Omron Sysmac Studio project RingBufferOpcUaExtensionLib (Sysmac Studio 1.63.0.7, LibraryProject)
(* Develop extension library for operating RingBuffer via OPC UA. *)

# Controller LIB: NX102-9000 version 1.64
Task Services (priority 18, period or condition 4000): ModelTest
Library RingBufferLib 0.0.2 (contents left out)

PROGRAM README
RETURN;
(*

# About this project
This project is for the development of `RingBufferOpcUaExtensionLib`.
`RingBufferOpcUaExtensionLib` exposes a **RingBuffer** using the FB instance publication of the OPC UA server.
The exposed **RingBuffer** can be used like an RPC with an appropriate OPC UA client and proper operating procedures.

## About programs

* POU/Program/ModelTest
  This is a test program for clients that use the exposed **RingBuffer**.


# このプロジェクトについて
このプロジェクトは、`RingBufferOpcUaExtensionLib`の開発用プロジェクトです。
`RingBufferOpcUaExtensionLib`は、OPC UAサーバのFBインスタンス公開を使用して`RingBuffer`を公開します。
公開した`RingBuffer`は、適切なOPC UAクライアントと操作手順によりRPCのように使用できるようになります。

## プログラムについて

* POU/プログラム/ModelTest
  公開した`RingBuffer`を使用するクライアント用のテストプログラムです。


For the parts to which I have rights, I follow POU/Program/LICENSE.
You are free to use and modify it, but we are not responsible for any damage or loss related to it.

(c) 2025 KITA Munemitsu

*)
END_PROGRAM

PROGRAM ModelTest
VAR
    ModelTestOpcUaRingBuffer : ModelTest_OpcUaRingBuffer;
END_VAR
IF P_First_Run THEN
	ModelTestOpcUaRingBuffer.Enable := TRUE;
END_IF;

ModelTestOpcUaRingBuffer();
END_PROGRAM

PROGRAM LICENSE
RETURN;
(*
The MIT License (MIT)

Copyright(c) 2025 KITA Munemitsu

Permission is hereby granted, free of charge, to any person obtaining a copy of this software and associated
documentation files (the “Software”), to deal in the Software without restriction, including without limitation
the rights to use, copy, modify, merge, publish, distribute, sublicense, and/or sell copies of the Software,
and to permit persons to whom the Software is furnished to do so, subject to the following conditions:

The above copyright notice and this permission notice shall be included in all copies or substantial portions of the Software.

THE SOFTWARE IS PROVIDED “AS IS”, WITHOUT WARRANTY OF ANY KIND, EXPRESS OR IMPLIED, INCLUDING BUT NOT
LIMITED TO THE WARRANTIES OF MERCHANTABILITY, FITNESS FOR A PARTICULAR PURPOSE AND NONINFRINGEMENT.
IN NO EVENT SHALL THE AUTHORS OR COPYRIGHT HOLDERS BE LIABLE FOR ANY CLAIM, DAMAGES OR OTHER LIABILITY,
WHETHER IN AN ACTION OF CONTRACT, TORT OR OTHERWISE, ARISING FROM, OUT OF OR IN CONNECTION WITH THE SOFTWARE
OR THE USE OR OTHER DEALINGS IN THE SOFTWARE.
*)
END_PROGRAM

FUNCTION_BLOCK stfreakjp\buf\extension\OpcUaRingBuffer
VAR
    Read : stfreakjp\buf\extension\OpcUaRingBuffer_read;
    ReadFully : stfreakjp\buf\extension\OpcUaRingBuffer_readFully;
    Peek : stfreakjp\buf\extension\OpcUaRingBuffer_peek;
    PeekFully : stfreakjp\buf\extension\OpcUaRingBuffer_peekFully;
    Write : stfreakjp\buf\extension\OpcUaRingBuffer_write;
    WriteFully : stfreakjp\buf\extension\OpcUaRingBuffer_writeFully;
    Consume : stfreakjp\buf\extension\OpcUaRingBuffer_consume;
    ClearBuffer : stfreakjp\buf\extension\OpcUaRingBuffer_clear;
    GetReadableSize : stfreakjp\buf\extension\OpcUaRingBuffer_getReadableSize;
    GetWritableSize : stfreakjp\buf\extension\OpcUaRingBuffer_getWritableSize;
    GetStat : stfreakjp\buf\extension\OpcUaRingBuffer_getStat;
    IsOverflow : stfreakjp\buf\extension\OpcUaRingBuffer_isOverflow;
    IsReadable : stfreakjp\buf\extension\OpcUaRingBuffer_isReadable;
    IsWritable : stfreakjp\buf\extension\OpcUaRingBuffer_isWritable;
    GetContext : stfreakjp\buf\extension\OpcUaRingBuffer_getContext;
    DiffWrite : stfreakjp\buf\extension\OpcUaRingBuffer_diffWrite;
    DiffRead : stfreakjp\buf\extension\OpcUaRingBuffer_diffRead;
    Diff : stfreakjp\buf\extension\OpcUaRingBuffer_diff;
    GetDiffStat : stfreakjp\buf\extension\OpcUaRingBuffer_getDiffStat;
END_VAR
VAR_INPUT
    Enable : BOOL;
END_VAR
VAR_IN_OUT
    BufferContext : stfreakjp\buf\RingBufferContext;
    Buffer : ARRAY[*] OF BYTE;
END_VAR
VAR_OUTPUT
    Busy : BOOL;
END_VAR
IF NOT (Enable OR Busy) THEN
	RETURN;
END_IF;

IF Enable <> Busy THEN
	Read.Execute := FALSE;
	ReadFully.Execute := FALSE;
	Peek.Execute := FALSE;
	PeekFully.Execute := FALSE;
	Write.Execute := FALSE;
	WriteFully.Execute := FALSE;
	Consume.Execute := FALSE;
	ClearBuffer.Execute := FALSE;
	GetReadableSize.Execute := FALSE;
	GetWritableSize.Execute := FALSE;
	GetStat.Execute := FALSE;
	IsOverflow.Execute := FALSE;
	IsReadable.Execute := FALSE;
	IsWritable.Execute := FALSE;
	
	GetContext.Execute := FALSE;
	DiffWrite.Execute := FALSE;
	DiffRead.Execute := FALSE;
	Diff.Execute := FALSE;
	GetDiffStat.Execute := FALSE;
END_IF;
Busy := Enable;

Read(BufferContext:=BufferContext, Buffer:=Buffer);
ReadFully(BufferContext:=BufferContext, Buffer:=Buffer);
Peek(BufferContext:=BufferContext, Buffer:=Buffer);
PeekFully(BufferContext:=BufferContext, Buffer:=Buffer);
Write(BufferContext:=BufferContext, Buffer:=Buffer);
WriteFully(BufferContext:=BufferContext, Buffer:=Buffer);
Consume(BufferContext:=BufferContext, Buffer:=Buffer);
ClearBuffer(BufferContext:=BufferContext, Buffer:=Buffer);
GetReadableSize(BufferContext:=BufferContext);
GetWritableSize(BufferContext:=BufferContext);
GetStat(BufferContext:=BufferContext);
IsOverflow(BufferContext:=BufferContext);
IsReadable(BufferContext:=BufferContext);
IsWritable(BufferContext:=BufferContext);
	
GetContext(BufferContext:=BufferContext);
DiffWrite(BufferContext:=BufferContext, Buffer:=Buffer);
DiffRead(BufferContext:=BufferContext, Buffer:=Buffer);
Diff(BufferContext:=BufferContext, Buffer:=Buffer);
GetDiffStat(BufferContext:=BufferContext);
END_FUNCTION_BLOCK

FUNCTION_BLOCK stfreakjp\buf\extension\OpcUaRingBuffer_read
VAR_INPUT
    Execute : BOOL := False;
END_VAR
VAR_IN_OUT
    BufferContext : stfreakjp\buf\RingBufferContext;
    Buffer : ARRAY[*] OF BYTE;
END_VAR
VAR_INPUT
    Size : UINT := 0;
END_VAR
VAR_OUTPUT
    Out : ARRAY[0..8191] OF BYTE;
    ReadSize : UINT;
    Overflow : BOOL;
    Done : BOOL;
END_VAR
IF NOT Execute THEN
	IF Done THEN
		ReadSize := 0;
		Overflow := FALSE;
		Done := FALSE;
	END_IF;
	
	RETURN;
END_IF;

IF Execute AND NOT Done THEN
	\\stfreakjp\buf\RingBuffer_read(
						Context:=BufferContext,
						Buffer:=Buffer,
						Size:=Size,
						Out:=Out,
						Head:=0,
						ReadSize=>ReadSize,
						Overflow=>Overflow);
	Done := TRUE;
END_IF;
END_FUNCTION_BLOCK

FUNCTION_BLOCK stfreakjp\buf\extension\OpcUaRingBuffer_readFully
VAR_INPUT
    Execute : BOOL;
END_VAR
VAR_IN_OUT
    BufferContext : stfreakjp\buf\RingBufferContext;
    Buffer : ARRAY[*] OF BYTE;
END_VAR
VAR_OUTPUT
    Out : ARRAY[0..8191] OF BYTE;
    ReadSize : UINT;
    Overflow : BOOL;
    Done : BOOL;
END_VAR
IF NOT Execute THEN
	IF Done THEN
		ReadSize := 0;
		Overflow := FALSE;
		Done := FALSE;
	END_IF;
	
	RETURN;
END_IF;

IF Execute AND NOT Done THEN
	\\stfreakjp\buf\RingBuffer_readFully(
						Context:=BufferContext,
						Buffer:=Buffer,
						Out:=Out,
						Head:=0,
						ReadSize=>ReadSize,
						Overflow=>Overflow);
	Done := TRUE;
END_IF;
END_FUNCTION_BLOCK

FUNCTION_BLOCK stfreakjp\buf\extension\OpcUaRingBuffer_peek
VAR_INPUT
    Execute : BOOL := False;
END_VAR
VAR_IN_OUT
    BufferContext : stfreakjp\buf\RingBufferContext;
    Buffer : ARRAY[*] OF BYTE;
END_VAR
VAR_INPUT
    Size : UINT := 0;
END_VAR
VAR_OUTPUT
    Out : ARRAY[0..8191] OF BYTE;
    ReadSize : UINT;
    Overflow : BOOL;
    Done : BOOL;
END_VAR
IF NOT Execute THEN
	IF Done THEN
		ReadSize := 0;
		Overflow := FALSE;
		Done := FALSE;
	END_IF;
	
	RETURN;
END_IF;

IF Execute AND NOT Done THEN
	\\stfreakjp\buf\RingBuffer_peek(
						Context:=BufferContext,
						Buffer:=Buffer,
						Size:=Size,
						Out:=Out,
						Head:=0,
						ReadSize=>ReadSize,
						Overflow=>Overflow);
	Done := TRUE;
END_IF;
END_FUNCTION_BLOCK

FUNCTION_BLOCK stfreakjp\buf\extension\OpcUaRingBuffer_peekFully
VAR_INPUT
    Execute : BOOL := False;
END_VAR
VAR_IN_OUT
    BufferContext : stfreakjp\buf\RingBufferContext;
    Buffer : ARRAY[*] OF BYTE;
END_VAR
VAR_OUTPUT
    Out : ARRAY[0..8191] OF BYTE;
    ReadSize : UINT;
    Overflow : BOOL;
    Done : BOOL;
END_VAR
IF NOT Execute THEN
	IF Done THEN
		ReadSize := 0;
		Overflow := FALSE;
		Done := FALSE;
	END_IF;
	
	RETURN;
END_IF;

IF Execute AND NOT Done THEN
	\\stfreakjp\buf\RingBuffer_peekFully(
						Context:=BufferContext,
						Buffer:=Buffer,
						Out:=Out,
						Head:=0,
						ReadSize=>ReadSize,
						Overflow=>Overflow);
	Done := TRUE;
END_IF;
END_FUNCTION_BLOCK

FUNCTION_BLOCK stfreakjp\buf\extension\OpcUaRingBuffer_write
VAR
    iTmpIn : ARRAY[0..8191] OF BYTE;
END_VAR
VAR_INPUT
    Execute : BOOL := False;
END_VAR
VAR_IN_OUT
    BufferContext : stfreakjp\buf\RingBufferContext;
    Buffer : ARRAY[*] OF BYTE;
END_VAR
VAR_INPUT
    In : ARRAY[0..8191] OF BYTE;
    Size : UINT := 0;
    AllowOverwrite : BOOL;
END_VAR
VAR_OUTPUT
    Ok : BOOL;
    Done : BOOL;
END_VAR
IF NOT Execute THEN
	Done := FALSE;

	RETURN;
END_IF;

IF Execute AND NOT Done THEN
	MemCopy(In:=In[0], AryOut:=iTmpIn[0], Size:=Size);	
	Ok := \\stfreakjp\buf\RingBuffer_write(
							  Context:=BufferContext,
							  Buffer:=Buffer,
							  In:=iTmpIn,
							  Head:=0,
							  Size:=Size,
							  AllowOverwrite:=AllowOverwrite);
	Done := TRUE;
END_IF;
END_FUNCTION_BLOCK

FUNCTION_BLOCK stfreakjp\buf\extension\OpcUaRingBuffer_writeFully
VAR
    iTmpIn : ARRAY[0..8191] OF BYTE;
END_VAR
VAR_INPUT
    Execute : BOOL := False;
END_VAR
VAR_IN_OUT
    BufferContext : stfreakjp\buf\RingBufferContext;
    Buffer : ARRAY[*] OF BYTE;
END_VAR
VAR_INPUT
    In : ARRAY[0..8191] OF BYTE;
    Size : UINT := 0;
END_VAR
VAR_OUTPUT
    WriteSize : UINT;
    Done : BOOL;
END_VAR
IF NOT Execute THEN
	IF Done THEN
		WriteSize := 0;
		Done := FALSE;
	END_IF;

	RETURN;
END_IF;

IF Execute AND NOT Done THEN
	MemCopy(In:=In[0], AryOut:=iTmpIn[0], Size:=Size);	
	\\stfreakjp\buf\RingBuffer_writeFully(
						Context:=BufferContext,
						Buffer:=Buffer,
						In:=iTmpIn,
						Head:=0,
						Size:=Size,
						WriteSize=>WriteSize);
	Done := TRUE;
END_IF;
END_FUNCTION_BLOCK

FUNCTION_BLOCK stfreakjp\buf\extension\OpcUaRingBuffer_consume
VAR_INPUT
    Execute : BOOL := False;
END_VAR
VAR_IN_OUT
    BufferContext : stfreakjp\buf\RingBufferContext;
    Buffer : ARRAY[*] OF BYTE;
END_VAR
VAR_INPUT
    Size : UINT := 0;
END_VAR
VAR_OUTPUT
    Ok : BOOL;
    Done : BOOL;
END_VAR
IF NOT Execute THEN
	Done := FALSE;
	
	RETURN;
END_IF;

IF Execute AND NOT Done THEN
	Ok := \\stfreakjp\buf\RingBuffer_consume(
							  Context:=BufferContext,
							  Buffer:=Buffer,
							  Size:=Size);
	Done := TRUE;
END_IF;
END_FUNCTION_BLOCK

FUNCTION_BLOCK stfreakjp\buf\extension\OpcUaRingBuffer_clear
VAR_INPUT
    Execute : BOOL := False;
END_VAR
VAR_IN_OUT
    BufferContext : stfreakjp\buf\RingBufferContext;
    Buffer : ARRAY[*] OF BYTE;
END_VAR
VAR_OUTPUT
    Ok : BOOL;
    Done : BOOL;
END_VAR
IF NOT Execute THEN
	Done := FALSE;
	
	RETURN;
END_IF;

IF Execute AND NOT Done THEN
	Ok := \\stfreakjp\buf\RingBuffer_clear(
							  Context:=BufferContext,
							  Buffer:=Buffer);
	Done := TRUE;
END_IF;
END_FUNCTION_BLOCK

FUNCTION_BLOCK stfreakjp\buf\extension\OpcUaRingBuffer_getReadableSize
VAR_INPUT
    Execute : BOOL := False;
END_VAR
VAR_IN_OUT
    BufferContext : stfreakjp\buf\RingBufferContext;
END_VAR
VAR_OUTPUT
    Size : UINT;
    Done : BOOL;
END_VAR
IF NOT Execute THEN
	IF Done THEN
		Size := 0;
		Done := FALSE;
	END_IF;
	
	RETURN;
END_IF;

IF Execute AND NOT Done THEN
	\\stfreakjp\buf\RingBuffer_getReadableSize(
						Context:=BufferContext,
						Size=>Size);
	Done := TRUE;
END_IF;
END_FUNCTION_BLOCK

FUNCTION_BLOCK stfreakjp\buf\extension\OpcUaRingBuffer_getWritableSize
VAR_INPUT
    Execute : BOOL;
END_VAR
VAR_IN_OUT
    BufferContext : stfreakjp\buf\RingBufferContext;
END_VAR
VAR_OUTPUT
    Size : UINT;
    Done : BOOL;
END_VAR
IF NOT Execute THEN
	IF Done THEN
		Size := 0;
		Done := FALSE;
	END_IF;
	
	RETURN;
END_IF;

IF Execute AND NOT Done THEN
	\\stfreakjp\buf\RingBuffer_getWritableSize(
						Context:=BufferContext,
						Size=>Size);
	Done := TRUE;
END_IF;
END_FUNCTION_BLOCK

FUNCTION_BLOCK stfreakjp\buf\extension\OpcUaRingBuffer_getStat
VAR_INPUT
    Execute : BOOL;
END_VAR
VAR_IN_OUT
    BufferContext : stfreakjp\buf\RingBufferContext;
END_VAR
VAR_OUTPUT
    WritableSize : UINT;
    ReadableSize : UINT;
    Overflow : BOOL;
    Done : BOOL;
END_VAR
IF NOT Execute THEN
	IF Done THEN
		WritableSize := 0;
		ReadableSize := 0;
		Overflow := FALSE;
		Done := FALSE;
	END_IF;
	
	RETURN;
END_IF;

IF Execute AND NOT Done THEN
	\\stfreakjp\buf\RingBuffer_getStat(
						Context:=BufferContext,
						WritableSize=>WritableSize,
						ReadableSize=>ReadableSize,
						Overflow=>Overflow);
	Done := TRUE;
END_IF;
END_FUNCTION_BLOCK

FUNCTION_BLOCK stfreakjp\buf\extension\OpcUaRingBuffer_isOverflow
VAR_INPUT
    Execute : BOOL;
END_VAR
VAR_IN_OUT
    BufferContext : stfreakjp\buf\RingBufferContext;
END_VAR
VAR_OUTPUT
    Overflow : BOOL;
    Done : BOOL;
END_VAR
IF NOT Execute THEN
	Overflow := FALSE;
	Done := FALSE;
	
	RETURN;
END_IF;

IF Execute AND NOT Done THEN
	Overflow := \\stfreakjp\buf\RingBuffer_isOverflow(
									Context:=BufferContext);
	Done := TRUE;
END_IF;
END_FUNCTION_BLOCK

FUNCTION_BLOCK stfreakjp\buf\extension\OpcUaRingBuffer_isReadable
VAR_INPUT
    Execute : BOOL;
END_VAR
VAR_IN_OUT
    BufferContext : stfreakjp\buf\RingBufferContext;
END_VAR
VAR_OUTPUT
    Readable : BOOL;
    Done : BOOL;
END_VAR
IF NOT Execute THEN
	Readable := FALSE;
	Done := FALSE;
	
	RETURN;
END_IF;

IF Execute AND NOT Done THEN
	Readable := \\stfreakjp\buf\RingBuffer_isReadable(
									Context:=BufferContext);
	Done := TRUE;
END_IF;
END_FUNCTION_BLOCK

FUNCTION_BLOCK stfreakjp\buf\extension\OpcUaRingBuffer_isWritable
VAR_INPUT
    Execute : BOOL;
END_VAR
VAR_IN_OUT
    BufferContext : stfreakjp\buf\RingBufferContext;
END_VAR
VAR_OUTPUT
    Writable : BOOL;
    Done : BOOL;
END_VAR
IF NOT Execute THEN
	Writable := FALSE;
	Done := FALSE;
	
	RETURN;
END_IF;

IF Execute AND NOT Done THEN
	Writable := \\stfreakjp\buf\RingBuffer_isWritable(
									Context:=BufferContext);
	Done := TRUE;
END_IF;
END_FUNCTION_BLOCK

FUNCTION_BLOCK stfreakjp\buf\extension\OpcUaRingBuffer_getContext
VAR_INPUT
    Execute : BOOL;
END_VAR
VAR_IN_OUT
    BufferContext : stfreakjp\buf\RingBufferContext;
END_VAR
VAR_OUTPUT
    Context : stfreakjp\buf\RingBufferContext;
    Done : BOOL;
END_VAR
IF NOT Execute THEN
	IF Done THEN
		Clear(Context);
		Done := FALSE;
	END_IF;
	
	RETURN;
END_IF;

IF Execute AND NOT Done THEN
	Context := BufferContext;
	Done := TRUE;
END_IF;
END_FUNCTION_BLOCK

FUNCTION_BLOCK stfreakjp\buf\extension\OpcUaRingBuffer_diffWrite
VAR
    iRefContext : stfreakjp\buf\RingBufferContext;
END_VAR
VAR_INPUT
    Execute : BOOL;
END_VAR
VAR_IN_OUT
    BufferContext : stfreakjp\buf\RingBufferContext;
    Buffer : ARRAY[*] OF BYTE;
END_VAR
VAR_INPUT
    RefContext : stfreakjp\buf\RingBufferContext;
END_VAR
VAR_OUTPUT
    Out : ARRAY[0..8191] OF BYTE;
    Size : UINT;
    Missing : BOOL;
    ComparedContext : stfreakjp\buf\RingBufferContext;
    Done : BOOL;
END_VAR
IF NOT Execute THEN
	IF Done THEN
		Size := 0;
		Missing := FALSE;
		Clear(ComparedContext);
		Done := FALSE;
	END_IF;
	
	RETURN;
END_IF;

IF Execute AND NOT Done THEN
	iRefContext := RefContext;
	\\stfreakjp\buf\RingBuffer_diffWrite(
						Context:=BufferContext,
						Buffer:=Buffer,
						RefContext:=iRefContext,
						Diff:=Out,
						Head:=0,
						Size=>Size,
						Missing=>Missing,
						ComparedContext=>ComparedContext);
	Done := TRUE;
END_IF;
END_FUNCTION_BLOCK

FUNCTION_BLOCK stfreakjp\buf\extension\OpcUaRingBuffer_diffRead
VAR
    iRefContext : stfreakjp\buf\RingBufferContext;
END_VAR
VAR_INPUT
    Execute : BOOL;
END_VAR
VAR_IN_OUT
    BufferContext : stfreakjp\buf\RingBufferContext;
    Buffer : ARRAY[*] OF BYTE;
END_VAR
VAR_INPUT
    RefContext : stfreakjp\buf\RingBufferContext;
END_VAR
VAR_OUTPUT
    Out : ARRAY[0..8191] OF BYTE;
    Size : UINT;
    Missing : BOOL;
    Overflow : BOOL;
    ComparedContext : stfreakjp\buf\RingBufferContext;
    Done : BOOL;
END_VAR
IF NOT Execute THEN
	IF Done THEN
		Size := 0;
		Missing := FALSE;
		Overflow := FALSE;
		Clear(ComparedContext);
		Done := FALSE;
	END_IF;
	
	RETURN;
END_IF;

IF Execute AND NOT Done THEN
	iRefContext := RefContext;
	\\stfreakjp\buf\RingBuffer_diffRead(
						Context:=BufferContext,
						Buffer:=Buffer,
						RefContext:=iRefContext,
						Diff:=Out,
						Head:=0,
						Size=>Size,
						Missing=>Missing,
						Overflow=>Overflow,
						ComparedContext=>ComparedContext);
	Done := TRUE;
END_IF;
END_FUNCTION_BLOCK

FUNCTION_BLOCK stfreakjp\buf\extension\OpcUaRingBuffer_diff
VAR
    iRefContext : stfreakjp\buf\RingBufferContext;
END_VAR
VAR_INPUT
    Execute : BOOL;
END_VAR
VAR_IN_OUT
    BufferContext : stfreakjp\buf\RingBufferContext;
    Buffer : ARRAY[*] OF BYTE;
END_VAR
VAR_INPUT
    RefContext : stfreakjp\buf\RingBufferContext;
END_VAR
VAR_OUTPUT
    DiffWrite : ARRAY[0..8191] OF BYTE;
    DiffWriteSize : UINT;
    DiffWriteMissing : BOOL;
    DiffWriteValid : BOOL;
    DiffRead : ARRAY[0..8191] OF BYTE;
    DiffReadSize : UINT;
    DiffReadMissing : BOOL;
    DiffReadValid : BOOL;
    Overflow : BOOL;
    ComparedContext : stfreakjp\buf\RingBufferContext;
    Done : BOOL;
END_VAR
IF NOT Execute THEN
	IF Done THEN
		DiffWriteSize := 0;
		DiffWriteMissing := FALSE;
		DiffWriteValid := FALSE;
		DiffReadSize := 0;
		DiffReadMissing := FALSE;
		DiffReadValid := FALSE;
		Overflow := FALSE;
		Done := FALSE;
	END_IF;
	
	RETURN;
END_IF;

IF Execute AND NOT Done THEN
	iRefContext := RefContext;
	\\stfreakjp\buf\RingBuffer_diff(
						Context:=BufferContext,
						Buffer:=Buffer,
						RefContext:=iRefContext,
						DiffWrite:=DiffWrite,
						DiffWriteHead:=0,
						DiffWriteSize=>DiffWriteSize,
						DiffWriteMissing=>DiffWriteMissing,
						DiffWriteValid=>DiffWriteValid,
						DiffRead:=DiffRead,
						DiffReadHead:=0,
						DiffReadSize=>DiffReadSize,
						DiffReadMissing=>DiffReadMissing,
						DiffReadValid=>DiffReadValid,
						Overflow=>Overflow,
						ComparedContext=>ComparedContext);
	Done := TRUE;
END_IF;
END_FUNCTION_BLOCK

FUNCTION_BLOCK stfreakjp\buf\extension\OpcUaRingBuffer_getDiffStat
VAR
    iRefContext : stfreakjp\buf\RingBufferContext;
END_VAR
VAR_INPUT
    Execute : BOOL;
END_VAR
VAR_IN_OUT
    BufferContext : stfreakjp\buf\RingBufferContext;
END_VAR
VAR_INPUT
    RefContext : stfreakjp\buf\RingBufferContext;
END_VAR
VAR_OUTPUT
    DiffWriteSize : UINT;
    DiffWriteMissing : BOOL;
    DiffReadSize : UINT;
    DiffReadMissing : BOOL;
    Overflow : BOOL;
    ComparedContext : stfreakjp\buf\RingBufferContext;
    Done : BOOL;
END_VAR
IF NOT Execute THEN
	IF Done THEN
		DiffWriteSize := 0;
		DiffWriteMissing := FALSE;
		DiffReadSize := 0;
		DiffReadMissing := FALSE;
		Overflow := FALSE;
		Clear(ComparedContext);
		Done := FALSE;
	END_IF;
	
	RETURN;
END_IF;

IF Execute AND NOT Done THEN
	iRefContext := RefContext;
	\\stfreakjp\buf\RingBuffer_getDiffStat(
						Context:=BufferContext,
						RefContext:=iRefContext,
						DiffWriteSize=>DiffWriteSize,
						DiffWriteMissing=>DiffWriteMissing,
						DiffReadSize=>DiffReadSize,
						DiffReadMissing=>DiffReadMissing,						
						Overflow=>Overflow,
						ComparedContext=>ComparedContext);
	Done := TRUE;
END_IF;
END_FUNCTION_BLOCK

FUNCTION_BLOCK ModelTest_OpcUaRingBuffer
VAR
    Target : stfreakjp\buf\extension\OpcUaRingBuffer;
    iBufferContext : stfreakjp\buf\RingBufferContext;
    iBuffer : ARRAY[0..65534] OF BYTE;
    Initialize : ModelTest_stateMethod;
    InitializeCount : UINT := 0;
    iInitializeContext : UINT := 0;
    TearDown : ModelTest_stateMethod;
    TearDownCount : UINT := 0;
    iTearDownContext : UINT := 0;
END_VAR
VAR_INPUT
    Enable : BOOL;
END_VAR
VAR_OUTPUT
    Busy : BOOL;
END_VAR
IF Enable AND NOT Busy THEN
	Initialize.Execute := FALSE;
	Clear(InitializeCount);
	TearDown.Execute := FALSE;
	Clear(TearDownCount);
	
	Clear(iBuffer);
	Clear(iBufferContext);
	\\stfreakjp\buf\RingBuffer_init(
						Context:=iBufferContext,
						Buffer:=iBuffer);
	Target.Enable := TRUE;
	
	Busy := TRUE;
ELSIF NOT Enable AND Busy THEN
	Initialize.Execute := FALSE;
	TearDown.Execute := FALSE;
	
	Target.Enable := FALSE;
	
	Busy := FALSE;	
END_IF;

IF Busy THEN
	Initialize(Context:=iInitializeContext);
	IF Initialize.Busy THEN
		CASE iInitializeContext OF
			// Init
			0:
				Clear(iBuffer);
				Clear(iBufferContext);
				\\stfreakjp\buf\RingBuffer_init(
									Context:=iBufferContext,
									Buffer:=iBuffer);
				Target.Enable := FALSE;
				
				Inc(iInitializeContext);
			1:
				Target.Enable := TRUE;

				iInitializeContext := 1000;
				
			// Done
			1000:
				Inc(InitializeCount);
				
				Inc(iInitializeContext);
		END_CASE;
	END_IF;

	TearDown(Context:=iTearDownContext);
	IF TearDown.Busy THEN
		CASE iTearDownContext OF
			// Init
			0:
				Clear(iBuffer);
				Clear(iBufferContext);
				\\stfreakjp\buf\RingBuffer_init(
									Context:=iBufferContext,
									Buffer:=iBuffer);
				
				iTearDownContext := 1000;
				
			// Done
			1000:
				Inc(TearDownCount);
			
				Inc(iTearDownContext);
		END_CASE;
	END_IF;
END_IF;

Target(BufferContext:=iBufferContext,
	   Buffer:=iBuffer);
END_FUNCTION_BLOCK

FUNCTION_BLOCK ModelTest_signalMethod
VAR_INPUT
    Execute : BOOL;
END_VAR
VAR_IN_OUT
    Context : BOOL;
END_VAR
VAR_OUTPUT
    Busy : BOOL;
    Done : BOOL;
END_VAR
IF Execute AND NOT Busy THEN
	Busy := TRUE;
ELSIF NOT Execute AND Busy THEN
	Context := FALSE;
	Busy := FALSE;
	Done := FALSE;
ELSIF Busy THEN
	Done := Context;
ELSIF NOT Execute THEN
	Context := FALSE;
	Done := FALSE;
END_IF;
END_FUNCTION_BLOCK

FUNCTION_BLOCK ModelTest_stateMethod
VAR_INPUT
    Execute : BOOL;
END_VAR
VAR_IN_OUT
    Context : UINT;
END_VAR
VAR_OUTPUT
    Busy : BOOL;
    Done : BOOL;
END_VAR
IF Execute AND NOT Busy THEN
	Busy := TRUE;
ELSIF NOT Execute AND Busy THEN
	Context := 0;
	Busy := FALSE;
	Done := FALSE;
ELSIF Busy THEN
	Done := Context >= 1000;
ELSIF NOT Execute THEN
	Context := 0;
	Done := FALSE;
END_IF;
END_FUNCTION_BLOCK